TYPE TcoInterpolatorControl :
STRUCT
	{attribute addProperty Name "<#Velocity Override#>"}
	Override : LREAL := 100.0;
	{attribute addProperty Name "<#Interpolation File#>"}
	FileName : STRING;
END_STRUCT
END_TYPE

(* stored: Version 1.1.0.1, ProductVersion 3.1.4024.12
   DUT TcoInterpolatorControl: Id {d19c6c08-ac03-00f7-135b-cc014fb5750a} *)
